(* IEC 61131-3 sources: stopGate_FuB/Logical/ProximityTestST, 5 files *)

(* ---- Types.typ ---- *)
TYPE

END_TYPE

(* ---- Cyclic.st ---- *)
PROGRAM _CYCLIC

	sensorST(inputSignal := inputSignal, onTimeDelay :=T#100ms , offTimeDelay := T#5000ms);

END_PROGRAM

(* ---- Exit.st ---- *)
PROGRAM _EXIT
	(* Insert code here *)

END_PROGRAM

(* ---- Init.st ---- *)
PROGRAM _INIT
	(* Insert code here *)

END_PROGRAM

(* ---- Variables.var ---- *)
VAR
	sensorST : onOffDebounce;
inputSignal : BOOL;
END_VAR
